DATA_BLOCK AutomatedDisassemblyLineDB
  VAR
    powerToolAvailable: BOOL := FALSE; // Input signal indicating the presence of a power tool on the line.
    disassemblyInspectionPassed: BOOL := FALSE; // Output signal indicating the status of disassembly process.
    cellIndicator: INT := 0; // A constant variable for cell identifier.
    powerToolData: STRUCT;
    (* A data structure for power tool's physical informtion.
    The structure is output of pre-processing stage;
    i.e., information from load cell, position sensor, vision system, etc
    is collected and stored into this variable.*)
    disassemblyPerformanceData: STRUCT;
    (* A data structure for disassembly process informtion.
    The structure is output of quality inspection of disassembly process.
    The variable can be used as an indicator of damage or defect level,
    as well as a feedback for tuning and improving robot performance.*)
    sortedComponents: INT;
    (*Output variable indicating the status of disassembled components.
    The variable is the result of sorting process,
    and can be used as a measure for seprating cells from non-cells components.*)
    cellData: STRUCT;
    (* A data structure for battery cell's informtion.
    The structure is output of classification stage;
    i.e., information from cell inspection, cell life test, etc
    is collected and stored into this variable.*)
  END_VAR
END_DATA_BLOCK

FUNCTION_BLOCK AutomatedDisassemblyLine
  METHODS
    CheckPowerToolPresence : BOOL;
    IdentifyPowerTool : STRUCT;
    DisassemblePowerTool(powerToolData: STRUCT) : BOOL, STRUCT;
    SortComponents : INT;
    InspectCellSpecification: STRUCT;
  END_METHODS

  METHODS IMPLEMENTATION
    CheckPowerToolPresence : BOOL
      (* Implement logic to check if there is a power tool available.*)
      RETURN powerToolAvailable;
    END_METHOD

    IdentifyPowerTool : STRUCT
      (* Implement logic for pre-processing stage; i.e. collecting object's information.*)
      RETURN powerToolData;
    END_METHOD

    DisassemblePowerTool(powerToolData: STRUCT) : BOOL, STRUCT
      (* Implement disassembly steps such as removing screws, openning the casing, extract the battery modules, etc.
      (* The method is an interface between the proccessing unit and the robot.*)
      RETURN disassemblyInspectionPassed, disassemblyPerformanceData;
    END_METHOD

    SortComponents : INT
      (* Implement sorting logic in order to identify the components.*)
      RETURN  sortedComponents;
    END_METHOD

    InspectCellSpecification: STRUCT
      (* Implement classification logic for battery cells.*)
      RETURN cellData;
    END_METHOD
  END_METHODS

  (* Main program *)
  // Check if a power tool is present on the line.
  CheckPowerToolPresence();
  // Start the pre-processing stage.
  IF powerToolAvailable THEN
    IdentifyPowerTool();
  END_IF;
  // Perform the disassembly process.
  DisassemblePowerTool(powerToolData);
  IF disassemblyInspectionPassed THEN
    // Performing the sorting process.
    SortComponents();
  END_IF;
  IF sortedComponents = cellIndicator THEN
    // Perform cell classification
    InspectCellSpecification();
  END_IF;
END_FUNCTION_BLOCK